% RSLogix 500 project Pump Control System with HOA Modes and Fault Protection.RSS, saved by version 8.30.00.16 %
PROJECT "UNTITLED"    % processor: Bul.1763 MicroLogix 1100 Series B %

PROGRAM FILES
  LAD 2 "MAIN"  5 rungs
  LAD 3 "IO"  8 rungs
  LAD 4 "CONTROLS"  11 rungs
  LAD 5 "FLOW ALARM"  4 rungs
  LAD 6 "PRES ALARM"  4 rungs

DATA FILES
  O0 OUTPUT  6 elements
  I1 INPUT  12 elements
  S2 STATUS  66 elements
  B3 BINARY  2 elements
  T4 TIMER  4 elements
  C5 COUNTER  1 elements
  R6 CONTROL  1 elements
  N7 INTEGER  4 elements
  F8 FLOAT  1 elements

LADDER 2 "MAIN"
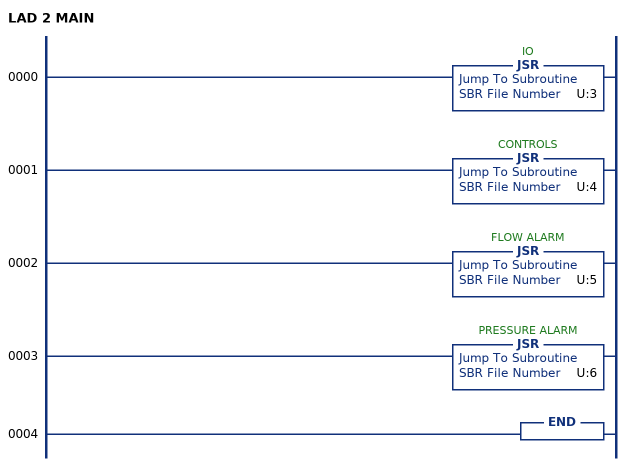
% Rung: 0 %
SOR JSR U:3 EOR
%   U:3  "IO" %
% Rung: 1 %
SOR JSR U:4 EOR
%   U:4  "CONTROLS" %
% Rung: 2 %
SOR JSR U:5 EOR
%   U:5  "FLOW ALARM" %
% Rung: 3 %
SOR JSR U:6 EOR
%   U:6  "PRESSURE ALARM" %
% Rung: 4 %
SOR END EOR

LADDER 3 "IO"
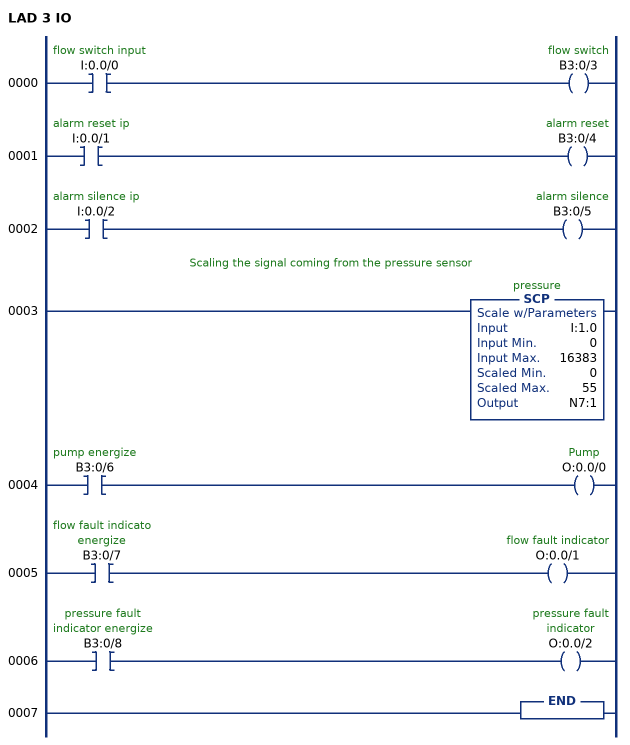
% Rung: 0 %
SOR XIC I:0.0/0 OTE B3:0/3 EOR
%   I:0.0/0  "flow switch input" %
%   B3:0/3  "flow switch" %
% Rung: 1 %
SOR XIC I:0.0/1 OTE B3:0/4 EOR
%   I:0.0/1  "alarm reset ip" %
%   B3:0/4  "alarm reset" %
% Rung: 2 %
SOR XIC I:0.0/2 OTE B3:0/5 EOR
%   I:0.0/2  "alarm silence ip" %
%   B3:0/5  "alarm silence" %
% Rung: 3 %
% Scaling the signal coming from the pressure sensor %
SOR SCP I:1.0 0 16383 0 55 N7:1 EOR
%   I:1.0  "pump pressure" %
%   N7:1  "pressure" %
% Rung: 4 %
SOR XIC B3:0/6 OTE O:0.0/0 EOR
%   B3:0/6  "pump energize" %
%   O:0.0/0  "Pump" %
% Rung: 5 %
SOR XIC B3:0/7 OTE O:0.0/1 EOR
%   B3:0/7  "flow fault indicato energize" %
%   O:0.0/1  "flow fault indicator" %
% Rung: 6 %
SOR XIC B3:0/8 OTE O:0.0/2 EOR
%   B3:0/8  "pressure fault indicator energize" %
%   O:0.0/2  "pressure fault indicator" %
% Rung: 7 %
SOR END EOR

LADDER 4 "CONTROLS"
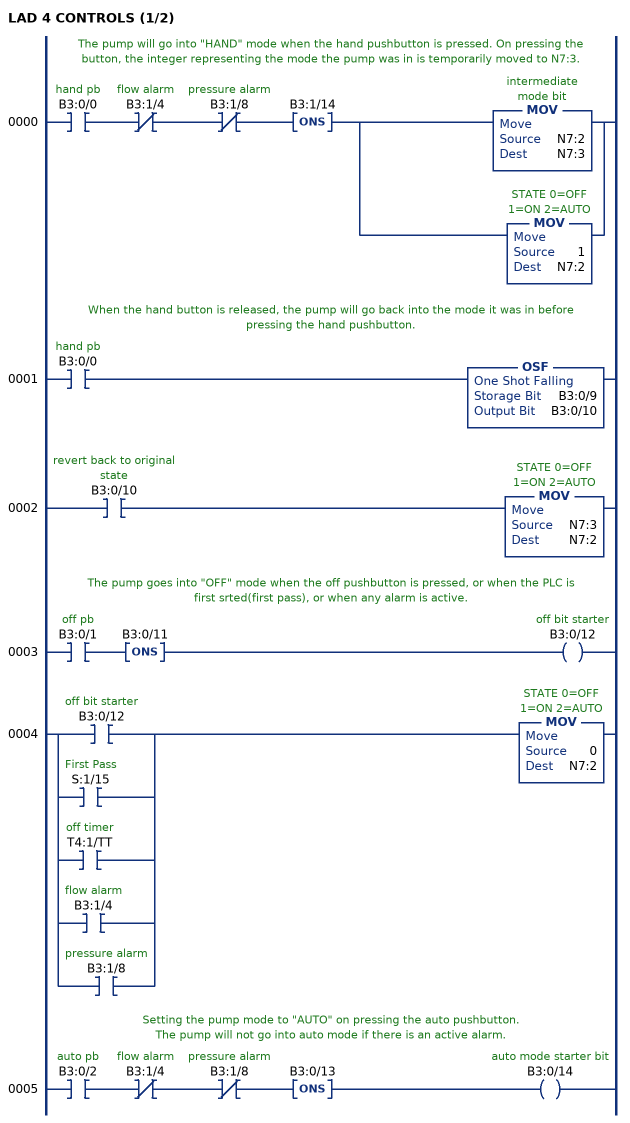
% Rung: 0 %
% The pump will go into "HAND" mode when the hand pushbutton is pressed. On pressing the button, the integer representing the mode the pump was in is temporarily moved to N7:3. %
SOR XIC B3:0/0 XIO B3:1/4 XIO B3:1/8 ONS B3:1/14 BST MOV N7:2 N7:3 NXB MOV 1 N7:2 BND EOR
%   B3:0/0  "hand pb" %
%   B3:1/4  "flow alarm" %
%   B3:1/8  "pressure alarm" %
%   N7:2  "STATE 0=OFF 1=ON 2=AUTO" %
%   N7:3  "intermediate mode bit" %
% Rung: 1 %
% When the hand button is released, the pump will go back into the mode it was in before pressing the hand pushbutton. %
SOR XIC B3:0/0 OSF B3:0/9 B3:0/10 EOR
%   B3:0/0  "hand pb" %
%   B3:0/10  "revert back to original state" %
% Rung: 2 %
SOR XIC B3:0/10 MOV N7:3 N7:2 EOR
%   B3:0/10  "revert back to original state" %
%   N7:3  "intermediate mode bit" %
%   N7:2  "STATE 0=OFF 1=ON 2=AUTO" %
% Rung: 3 %
% The pump goes into "OFF" mode when the off pushbutton is pressed, or when the PLC is first srted(first pass), or when any alarm is active. %
SOR XIC B3:0/1 ONS B3:0/11 OTE B3:0/12 EOR
%   B3:0/1  "off pb" %
%   B3:0/12  "off bit starter" %
% Rung: 4 %
SOR BST XIC B3:0/12 NXB XIC S:1/15 NXB XIC T4:1/TT NXB XIC B3:1/4 NXB XIC B3:1/8 BND MOV 0 N7:2 EOR
%   B3:0/12  "off bit starter" %
%   S:1/15  "First Pass" %
%   T4:1  "off timer" %
%   B3:1/4  "flow alarm" %
%   B3:1/8  "pressure alarm" %
%   N7:2  "STATE 0=OFF 1=ON 2=AUTO" %
% Rung: 5 %
% Setting the pump mode to "AUTO" on pressing the auto pushbutton.
% The pump will not go into auto mode if there is an active alarm. %
SOR XIC B3:0/2 XIO B3:1/4 XIO B3:1/8 ONS B3:0/13 OTE B3:0/14 EOR
%   B3:0/2  "auto pb" %
%   B3:1/4  "flow alarm" %
%   B3:1/8  "pressure alarm" %
%   B3:0/14  "auto mode starter bit" %

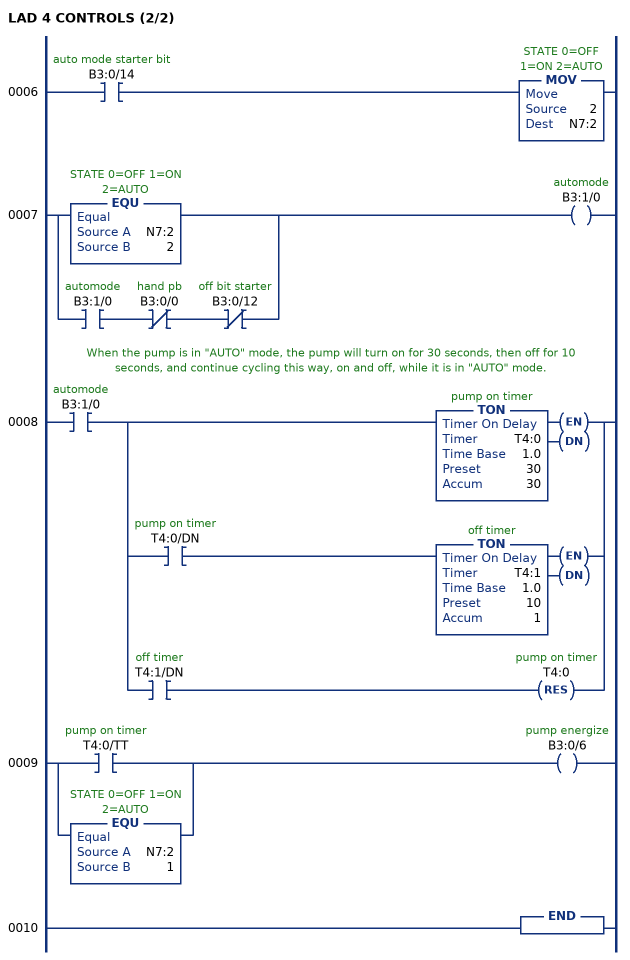
% Rung: 6 %
SOR XIC B3:0/14 MOV 2 N7:2 EOR
%   B3:0/14  "auto mode starter bit" %
%   N7:2  "STATE 0=OFF 1=ON 2=AUTO" %
% Rung: 7 %
SOR BST EQU N7:2 2 NXB XIC B3:1/0 XIO B3:0/0 XIO B3:0/12 BND OTE B3:1/0 EOR
%   N7:2  "STATE 0=OFF 1=ON 2=AUTO" %
%   B3:1/0  "automode" %
%   B3:0/0  "hand pb" %
%   B3:0/12  "off bit starter" %
% Rung: 8 %
% When the pump is in "AUTO" mode, the pump will turn on for 30 seconds, then off for 10 seconds, and continue cycling this way, on and off, while it is in "AUTO" mode. %
SOR XIC B3:1/0 BST TON T4:0 1.0 30 30 NXB XIC T4:0/DN TON T4:1 1.0 10 1 NXB XIC T4:1/DN RES T4:0 BND EOR
%   B3:1/0  "automode" %
%   T4:0  "pump on timer" %
%   T4:1  "off timer" %
% Rung: 9 %
SOR BST XIC T4:0/TT NXB EQU N7:2 1 BND OTE B3:0/6 EOR
%   T4:0  "pump on timer" %
%   N7:2  "STATE 0=OFF 1=ON 2=AUTO" %
%   B3:0/6  "pump energize" %
% Rung: 10 %
SOR END EOR

LADDER 5 "FLOW ALARM"
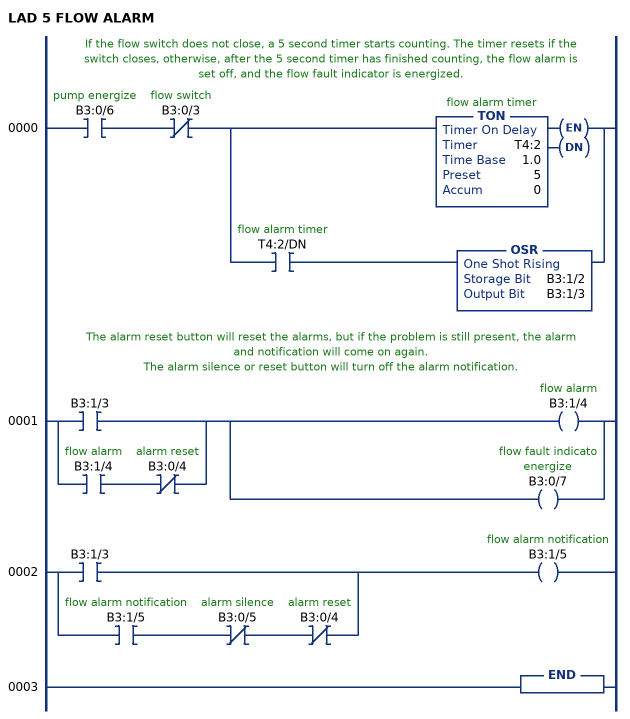
% Rung: 0 %
% If the flow switch does not close, a 5 second timer starts counting. The timer resets if the switch closes, otherwise, after the 5 second timer has finished counting, the flow alarm is set off, and the flow fault indicator is energized. %
SOR XIC B3:0/6 XIO B3:0/3 BST TON T4:2 1.0 5 0 NXB XIC T4:2/DN OSR B3:1/2 B3:1/3 BND EOR
%   B3:0/6  "pump energize" %
%   B3:0/3  "flow switch" %
%   T4:2  "flow alarm timer" %
% Rung: 1 %
% The alarm reset button will reset the alarms, but if the problem is still present, the alarm and notification will come on again.
% The alarm silence or reset button will turn off the alarm notification. %
SOR BST XIC B3:1/3 NXB XIC B3:1/4 XIO B3:0/4 BND BST OTE B3:1/4 NXB OTE B3:0/7 BND EOR
%   B3:1/4  "flow alarm" %
%   B3:0/4  "alarm reset" %
%   B3:0/7  "flow fault indicato energize" %
% Rung: 2 %
SOR BST XIC B3:1/3 NXB XIC B3:1/5 XIO B3:0/5 XIO B3:0/4 BND OTE B3:1/5 EOR
%   B3:1/5  "flow alarm notification" %
%   B3:0/5  "alarm silence" %
%   B3:0/4  "alarm reset" %
% Rung: 3 %
SOR END EOR

LADDER 6 "PRES ALARM"
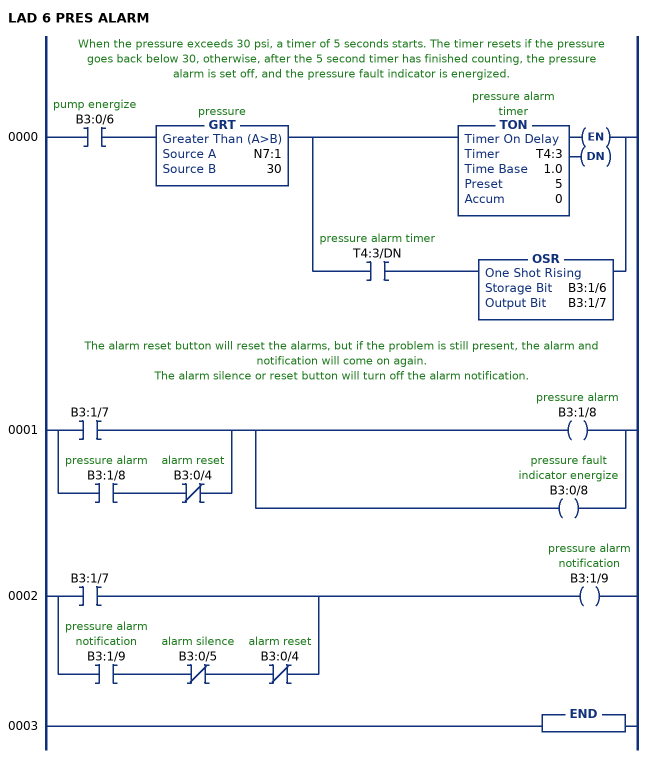
% Rung: 0 %
% When the pressure exceeds 30 psi, a timer of 5 seconds starts. The timer resets if the pressure goes back below 30, otherwise, after the 5 second timer has finished counting, the pressure alarm is set off, and the pressure fault indicator is energized. %
SOR XIC B3:0/6 GRT N7:1 30 BST TON T4:3 1.0 5 0 NXB XIC T4:3/DN OSR B3:1/6 B3:1/7 BND EOR
%   B3:0/6  "pump energize" %
%   N7:1  "pressure" %
%   T4:3  "pressure alarm timer" %
% Rung: 1 %
% The alarm reset button will reset the alarms, but if the problem is still present, the alarm and notification will come on again.
% The alarm silence or reset button will turn off the alarm notification. %
SOR BST XIC B3:1/7 NXB XIC B3:1/8 XIO B3:0/4 BND BST OTE B3:1/8 NXB OTE B3:0/8 BND EOR
%   B3:1/8  "pressure alarm" %
%   B3:0/4  "alarm reset" %
%   B3:0/8  "pressure fault indicator energize" %
% Rung: 2 %
SOR BST XIC B3:1/7 NXB XIC B3:1/9 XIO B3:0/5 XIO B3:0/4 BND OTE B3:1/9 EOR
%   B3:1/9  "pressure alarm notification" %
%   B3:0/5  "alarm silence" %
%   B3:0/4  "alarm reset" %
% Rung: 3 %
SOR END EOR

OTHER DOCUMENTED ADDRESSES
  B3:0/15  "auto mode energizer"
  B3:1/1  "handmode"
  N7:0  "prssure sensor input"

COMMENTS NOT ATTACHED TO A CURRENT RUNG
  N7:1: Scaling the signal coming from the pressure sensor

DATA TABLE (non-zero values as saved)
DATA B3
% B3:0 % 0X0008 0X0001
DATA T4
% .PRE .ACC %
% T4:0 % 30 30
% T4:1 % 10 1
% T4:2 % 5 0
% T4:3 % 5 0
DATA N7
% N7:0 % 8000 27 0 0
